{attribute 'GeneratedUsingTerminal: EK1122-0000-0018'}
{attribute addProperty BoxType "EK1122-0000-0018"}
{attribute addProperty Id "Beckhoff_ER3xxxsub_EK1100EK1100_1FC0878B2A_0001_ER3174_0002_0016ER3174_BE8A5C9E44A_0002_ER3174_0002_0022ER3174_BE8A5C9E44A_0003_ER3174_0002_0023ER3174_BE8A5C9E44A_0004_ER3184_0002_0019ER3184_BE8A5C9E44A_0005_ER3184_0002_0020ER3184_BE8A5C9E44A_0006_ER3184_0002_0021ER3184_BE8A5C9E44A_0007_ER3184_1002_0020ER3184_BE8A5C9E44A_0008_ER3184_1002_0021ER3184_BE8A5C9E44A_0009_ER3204_0002_0016ER3204_0999352444A_0010_ER3204_0002_0020ER3204_0999352444A_0011_ER3204_0002_0021ER3204_5F3CD6E040A_0012_ER3314_0002_0021ER3314_0E0DF94E40"}
{attribute addProperty CRC "4099995439"}
{attribute addProperty Size "522"}
TYPE Beckhoff_ER3xxxEK1122_F460F72F EXTENDS EK1122_1FC0878B :
STRUCT
	{attribute addProperty Name "Beckhoff_ER3xxxsub_EK1100"}
	{attribute addProperty PreviousPort "Beckhoff ER3xxxEK1122 : D"}
	Beckhoff_ER3xxxsub_EK1100 : EK1100_1FC0878B;
	{attribute addProperty Name "A_0001_ER3174_0002_0016"}
	{attribute addProperty PreviousPort "Beckhoff ER3xxxsub EK1100 : C"}
	A_0001_ER3174_0002_0016 : ER3174_BE8A5C9E;
	{attribute addProperty Name "A_0002_ER3174_0002_0022"}
	{attribute addProperty PreviousPort "A_0001(ER3174-0002-0016) : B"}
	A_0002_ER3174_0002_0022 : ER3174_BE8A5C9E;
	{attribute addProperty Name "A_0003_ER3174_0002_0023"}
	{attribute addProperty PreviousPort "A_0002(ER3174-0002-0022) : B"}
	A_0003_ER3174_0002_0023 : ER3174_BE8A5C9E;
	{attribute addProperty Name "A_0004_ER3184_0002_0019"}
	{attribute addProperty PreviousPort "A_0003(ER3174-0002-0023) : B"}
	A_0004_ER3184_0002_0019 : ER3184_BE8A5C9E;
	{attribute addProperty Name "A_0005_ER3184_0002_0020"}
	{attribute addProperty PreviousPort "A_0004(ER3184-0002-0019) : B"}
	A_0005_ER3184_0002_0020 : ER3184_BE8A5C9E;
	{attribute addProperty Name "A_0006_ER3184_0002_0021"}
	{attribute addProperty PreviousPort "A_0005(ER3184-0002-0020) : B"}
	A_0006_ER3184_0002_0021 : ER3184_BE8A5C9E;
	{attribute addProperty Name "A_0007_ER3184_1002_0020"}
	{attribute addProperty PreviousPort "A_0006(ER3184-0002-0021) : B"}
	A_0007_ER3184_1002_0020 : ER3184_BE8A5C9E;
	{attribute addProperty Name "A_0008_ER3184_1002_0021"}
	{attribute addProperty PreviousPort "A_0007(ER3184-1002-0020) : B"}
	A_0008_ER3184_1002_0021 : ER3184_BE8A5C9E;
	{attribute addProperty Name "A_0009_ER3204_0002_0016"}
	{attribute addProperty PreviousPort "A_0008(ER3184-1002-0021) : B"}
	A_0009_ER3204_0002_0016 : ER3204_09993524;
	{attribute addProperty Name "A_0010_ER3204_0002_0020"}
	{attribute addProperty PreviousPort "A_0009(ER3204-0002-0016) : B"}
	A_0010_ER3204_0002_0020 : ER3204_09993524;
	{attribute addProperty Name "A_0011_ER3204_0002_0021"}
	{attribute addProperty PreviousPort "A_0010(ER3204-0002-0020) : B"}
	A_0011_ER3204_0002_0021 : ER3204_5F3CD6E0;
	{attribute addProperty Name "A_0012_ER3314_0002_0021"}
	{attribute addProperty PreviousPort "A_0011(ER3204-0002-0021) : B"}
	A_0012_ER3314_0002_0021 : ER3314_0E0DF94E;
END_STRUCT
END_TYPE

(* stored: Version 1.2.0.0, ProductVersion 3.1.4024.9
   DUT Beckhoff_ER3xxxEK1122_F460F72F: Id {f93ac431-be9e-4ed3-b334-0b3a33b01ca8} *)
